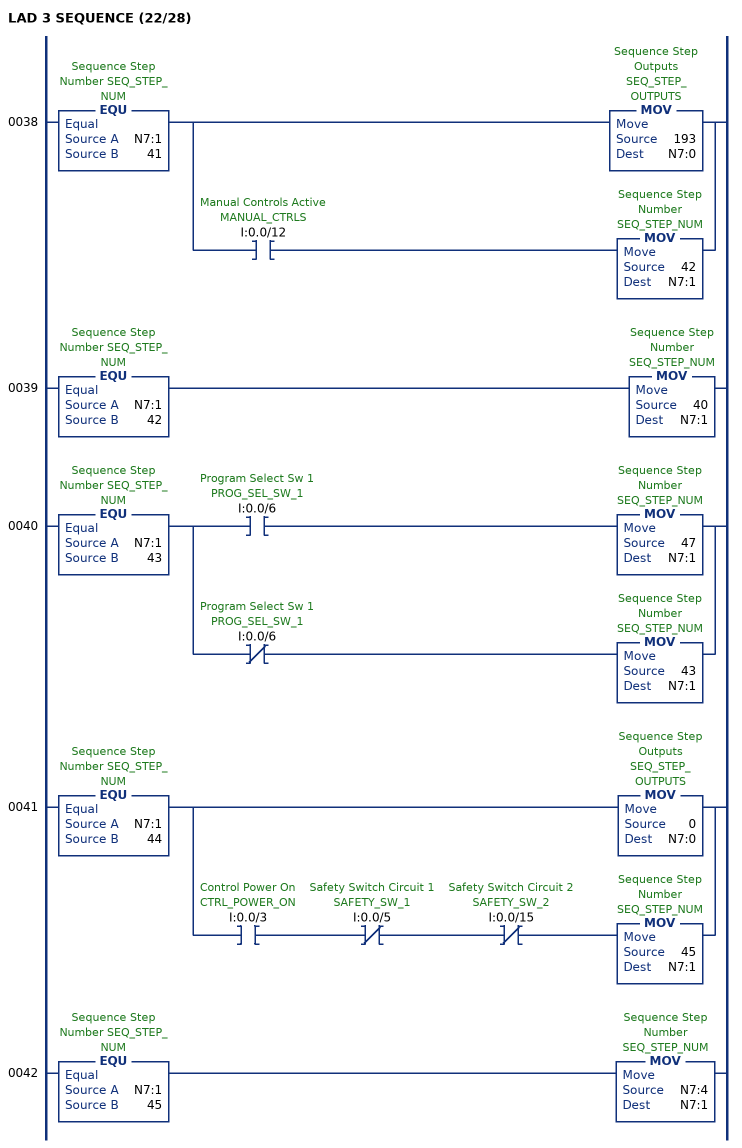
% Rung: 38 %
SOR EQU N7:1 41 BST MOV 193 N7:0 NXB XIC I:0.0/12 MOV 42 N7:1 BND EOR
%   N7:1  SEQ_STEP_NUM  "Sequence Step Number" %
%   N7:0  SEQ_STEP_OUTPUTS  "Sequence Step Outputs" %
%   I:0.0/12  MANUAL_CTRLS  "Manual Controls Active" %
% Rung: 39 %
SOR EQU N7:1 42 MOV 40 N7:1 EOR
%   N7:1  SEQ_STEP_NUM  "Sequence Step Number" %
% Rung: 40 %
SOR EQU N7:1 43 BST XIC I:0.0/6 MOV 47 N7:1 NXB XIO I:0.0/6 MOV 43 N7:1 BND EOR
%   N7:1  SEQ_STEP_NUM  "Sequence Step Number" %
%   I:0.0/6  PROG_SEL_SW_1  "Program Select Sw 1" %
% Rung: 41 %
SOR EQU N7:1 44 BST MOV 0 N7:0 NXB XIC I:0.0/3 XIO I:0.0/5 XIO I:0.0/15 MOV 45 N7:1 BND EOR
%   N7:1  SEQ_STEP_NUM  "Sequence Step Number" %
%   N7:0  SEQ_STEP_OUTPUTS  "Sequence Step Outputs" %
%   I:0.0/3  CTRL_POWER_ON  "Control Power On" %
%   I:0.0/5  SAFETY_SW_1  "Safety Switch Circuit 1" %
%   I:0.0/15  SAFETY_SW_2  "Safety Switch Circuit 2" %
% Rung: 42 %
SOR EQU N7:1 45 MOV N7:4 N7:1 EOR
%   N7:1  SEQ_STEP_NUM  "Sequence Step Number" %
%   N7:4  STORED_SEQ_STEP  "Stored Sequence Step" %

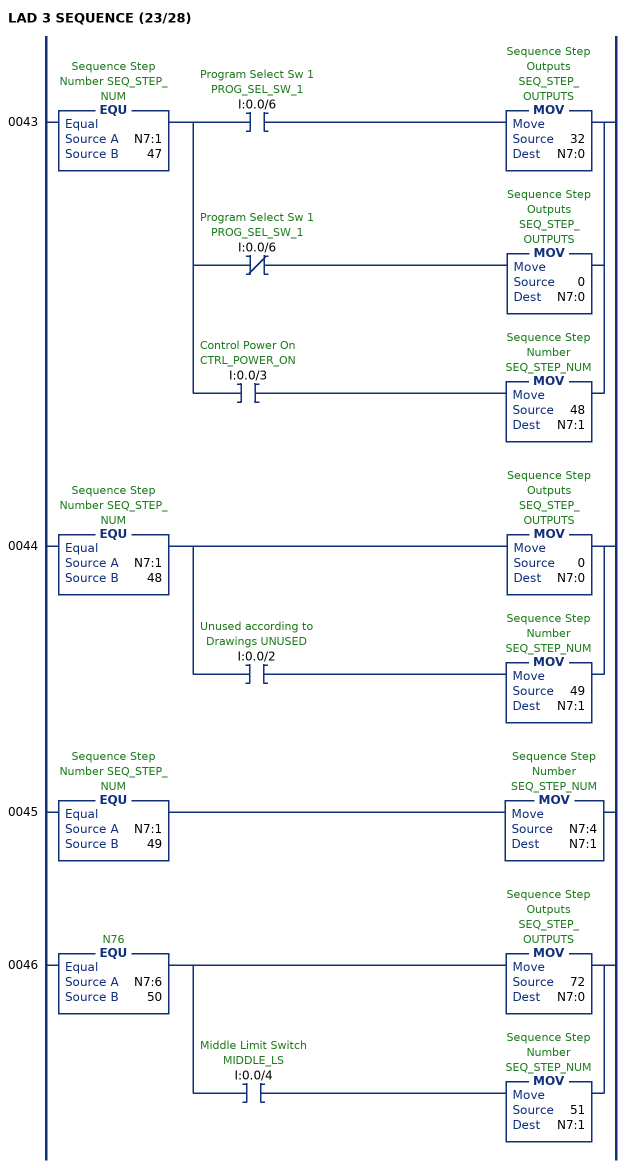
% Rung: 43 %
SOR EQU N7:1 47 BST XIC I:0.0/6 MOV 32 N7:0 NXB XIO I:0.0/6 MOV 0 N7:0 NXB XIC I:0.0/3 MOV 48 N7:1 BND EOR
%   N7:1  SEQ_STEP_NUM  "Sequence Step Number" %
%   I:0.0/6  PROG_SEL_SW_1  "Program Select Sw 1" %
%   N7:0  SEQ_STEP_OUTPUTS  "Sequence Step Outputs" %
%   I:0.0/3  CTRL_POWER_ON  "Control Power On" %
% Rung: 44 %
SOR EQU N7:1 48 BST MOV 0 N7:0 NXB XIC I:0.0/2 MOV 49 N7:1 BND EOR
%   N7:1  SEQ_STEP_NUM  "Sequence Step Number" %
%   N7:0  SEQ_STEP_OUTPUTS  "Sequence Step Outputs" %
%   I:0.0/2  UNUSED  "Unused according to Drawings" %
% Rung: 45 %
SOR EQU N7:1 49 MOV N7:4 N7:1 EOR
%   N7:1  SEQ_STEP_NUM  "Sequence Step Number" %
%   N7:4  STORED_SEQ_STEP  "Stored Sequence Step" %
% Rung: 46 %
SOR EQU N7:6 50 BST MOV 72 N7:0 NXB XIC I:0.0/4 MOV 51 N7:1 BND EOR
%   N7:6  N76 %
%   N7:0  SEQ_STEP_OUTPUTS  "Sequence Step Outputs" %
%   I:0.0/4  MIDDLE_LS  "Middle Limit Switch" %
%   N7:1  SEQ_STEP_NUM  "Sequence Step Number" %

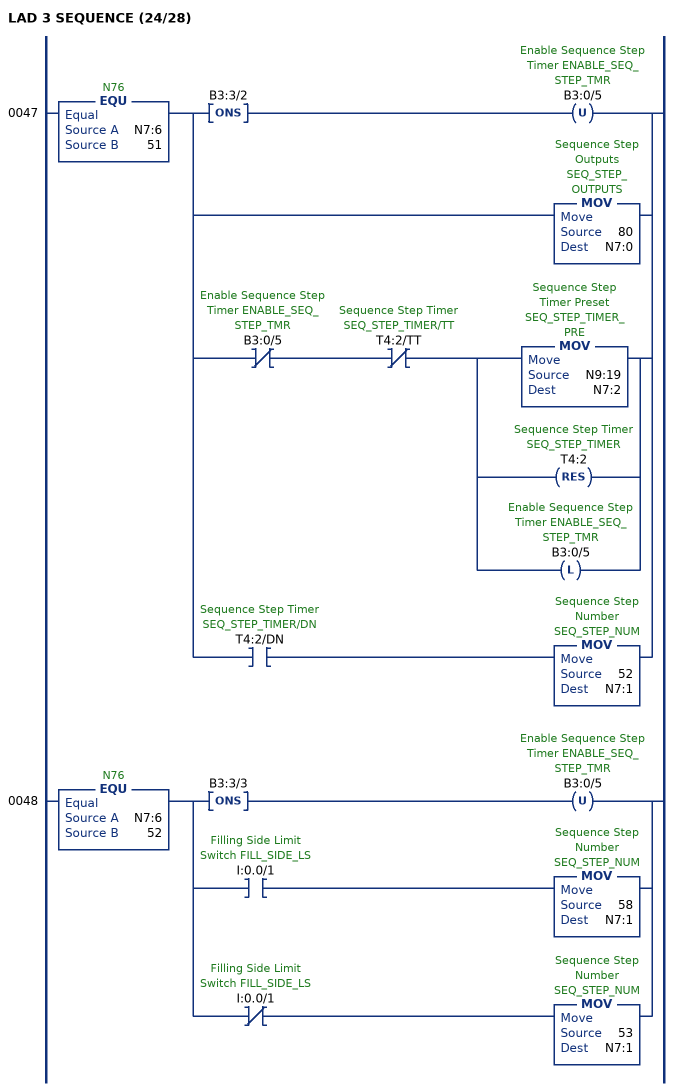
% Rung: 47 %
SOR EQU N7:6 51 BST ONS B3:3/2 OTU B3:0/5 NXB MOV 80 N7:0 NXB XIO B3:0/5 XIO T4:2/TT BST MOV N9:19 N7:2 NXB RES T4:2 NXB OTL B3:0/5 BND NXB XIC T4:2/DN MOV 52 N7:1 BND EOR
%   N7:6  N76 %
%   B3:0/5  ENABLE_SEQ_STEP_TMR  "Enable Sequence Step Timer" %
%   N7:0  SEQ_STEP_OUTPUTS  "Sequence Step Outputs" %
%   T4:2  SEQ_STEP_TIMER  "Sequence Step Timer" %
%   N7:2  SEQ_STEP_TIMER_PRE  "Sequence Step Timer Preset" %
%   N7:1  SEQ_STEP_NUM  "Sequence Step Number" %
% Rung: 48 %
SOR EQU N7:6 52 BST ONS B3:3/3 OTU B3:0/5 NXB XIC I:0.0/1 MOV 58 N7:1 NXB XIO I:0.0/1 MOV 53 N7:1 BND EOR
%   N7:6  N76 %
%   B3:0/5  ENABLE_SEQ_STEP_TMR  "Enable Sequence Step Timer" %
%   I:0.0/1  FILL_SIDE_LS  "Filling Side Limit Switch" %
%   N7:1  SEQ_STEP_NUM  "Sequence Step Number" %

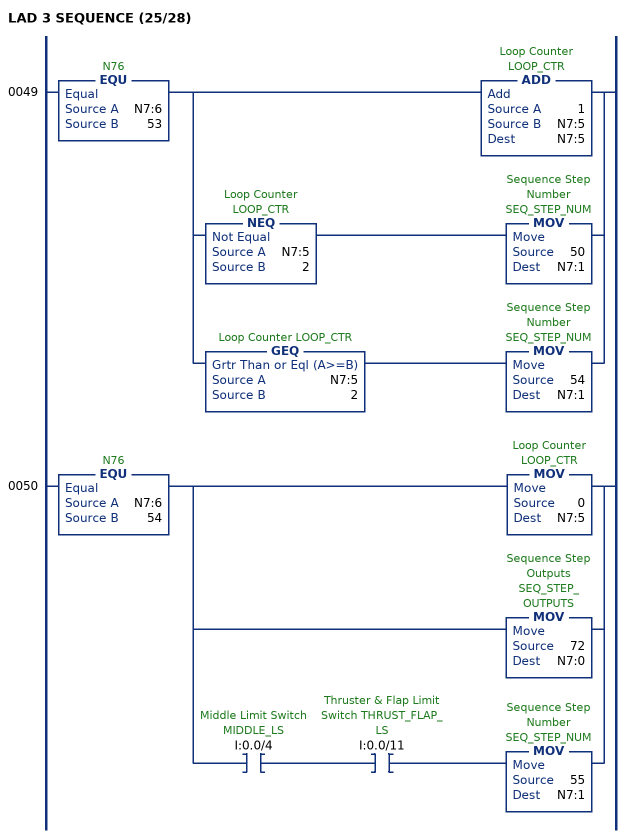
% Rung: 49 %
SOR EQU N7:6 53 BST ADD 1 N7:5 N7:5 NXB NEQ N7:5 2 MOV 50 N7:1 NXB GEQ N7:5 2 MOV 54 N7:1 BND EOR
%   N7:6  N76 %
%   N7:5  LOOP_CTR  "Loop Counter" %
%   N7:1  SEQ_STEP_NUM  "Sequence Step Number" %
% Rung: 50 %
SOR EQU N7:6 54 BST MOV 0 N7:5 NXB MOV 72 N7:0 NXB XIC I:0.0/4 XIC I:0.0/11 MOV 55 N7:1 BND EOR
%   N7:6  N76 %
%   N7:5  LOOP_CTR  "Loop Counter" %
%   N7:0  SEQ_STEP_OUTPUTS  "Sequence Step Outputs" %
%   I:0.0/4  MIDDLE_LS  "Middle Limit Switch" %
%   I:0.0/11  THRUST_FLAP_LS  "Thruster & Flap Limit Switch" %
%   N7:1  SEQ_STEP_NUM  "Sequence Step Number" %

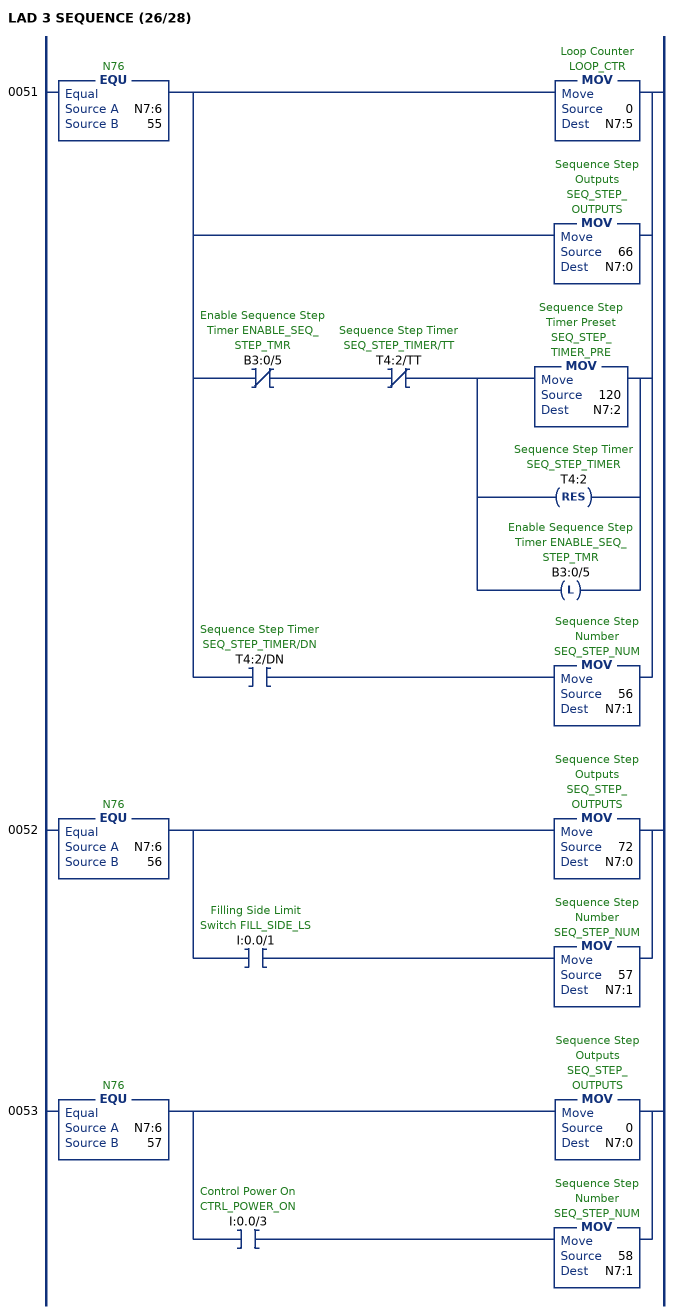
% Rung: 51 %
SOR EQU N7:6 55 BST MOV 0 N7:5 NXB MOV 66 N7:0 NXB XIO B3:0/5 XIO T4:2/TT BST MOV 120 N7:2 NXB RES T4:2 NXB OTL B3:0/5 BND NXB XIC T4:2/DN MOV 56 N7:1 BND EOR
%   N7:6  N76 %
%   N7:5  LOOP_CTR  "Loop Counter" %
%   N7:0  SEQ_STEP_OUTPUTS  "Sequence Step Outputs" %
%   B3:0/5  ENABLE_SEQ_STEP_TMR  "Enable Sequence Step Timer" %
%   T4:2  SEQ_STEP_TIMER  "Sequence Step Timer" %
%   N7:2  SEQ_STEP_TIMER_PRE  "Sequence Step Timer Preset" %
%   N7:1  SEQ_STEP_NUM  "Sequence Step Number" %
% Rung: 52 %
SOR EQU N7:6 56 BST MOV 72 N7:0 NXB XIC I:0.0/1 MOV 57 N7:1 BND EOR
%   N7:6  N76 %
%   N7:0  SEQ_STEP_OUTPUTS  "Sequence Step Outputs" %
%   I:0.0/1  FILL_SIDE_LS  "Filling Side Limit Switch" %
%   N7:1  SEQ_STEP_NUM  "Sequence Step Number" %
% Rung: 53 %
SOR EQU N7:6 57 BST MOV 0 N7:0 NXB XIC I:0.0/3 MOV 58 N7:1 BND EOR
%   N7:6  N76 %
%   N7:0  SEQ_STEP_OUTPUTS  "Sequence Step Outputs" %
%   I:0.0/3  CTRL_POWER_ON  "Control Power On" %
%   N7:1  SEQ_STEP_NUM  "Sequence Step Number" %

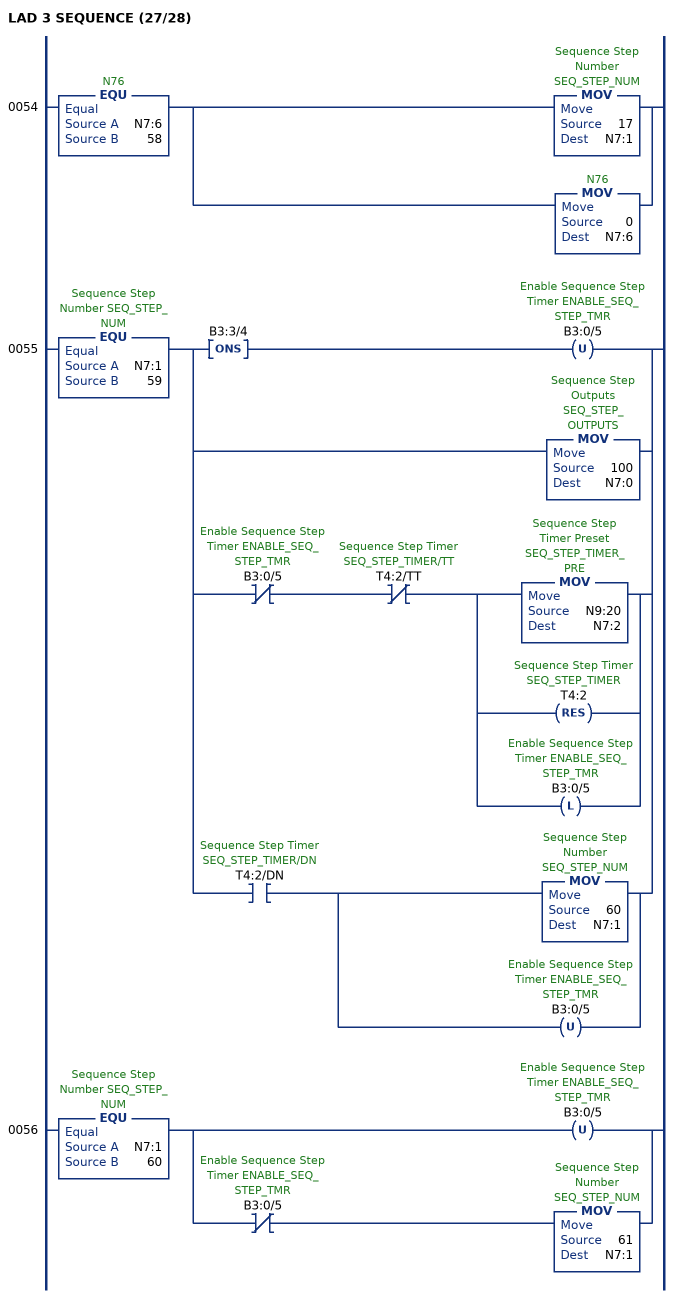
% Rung: 54 %
SOR EQU N7:6 58 BST MOV 17 N7:1 NXB MOV 0 N7:6 BND EOR
%   N7:6  N76 %
%   N7:1  SEQ_STEP_NUM  "Sequence Step Number" %
% Rung: 55 %
SOR EQU N7:1 59 BST ONS B3:3/4 OTU B3:0/5 NXB MOV 100 N7:0 NXB XIO B3:0/5 XIO T4:2/TT BST MOV N9:20 N7:2 NXB RES T4:2 NXB OTL B3:0/5 BND NXB XIC T4:2/DN BST MOV 60 N7:1 NXB OTU B3:0/5 BND BND EOR
%   N7:1  SEQ_STEP_NUM  "Sequence Step Number" %
%   B3:0/5  ENABLE_SEQ_STEP_TMR  "Enable Sequence Step Timer" %
%   N7:0  SEQ_STEP_OUTPUTS  "Sequence Step Outputs" %
%   T4:2  SEQ_STEP_TIMER  "Sequence Step Timer" %
%   N7:2  SEQ_STEP_TIMER_PRE  "Sequence Step Timer Preset" %
% Rung: 56 %
SOR EQU N7:1 60 BST OTU B3:0/5 NXB XIO B3:0/5 MOV 61 N7:1 BND EOR
%   N7:1  SEQ_STEP_NUM  "Sequence Step Number" %
%   B3:0/5  ENABLE_SEQ_STEP_TMR  "Enable Sequence Step Timer" %

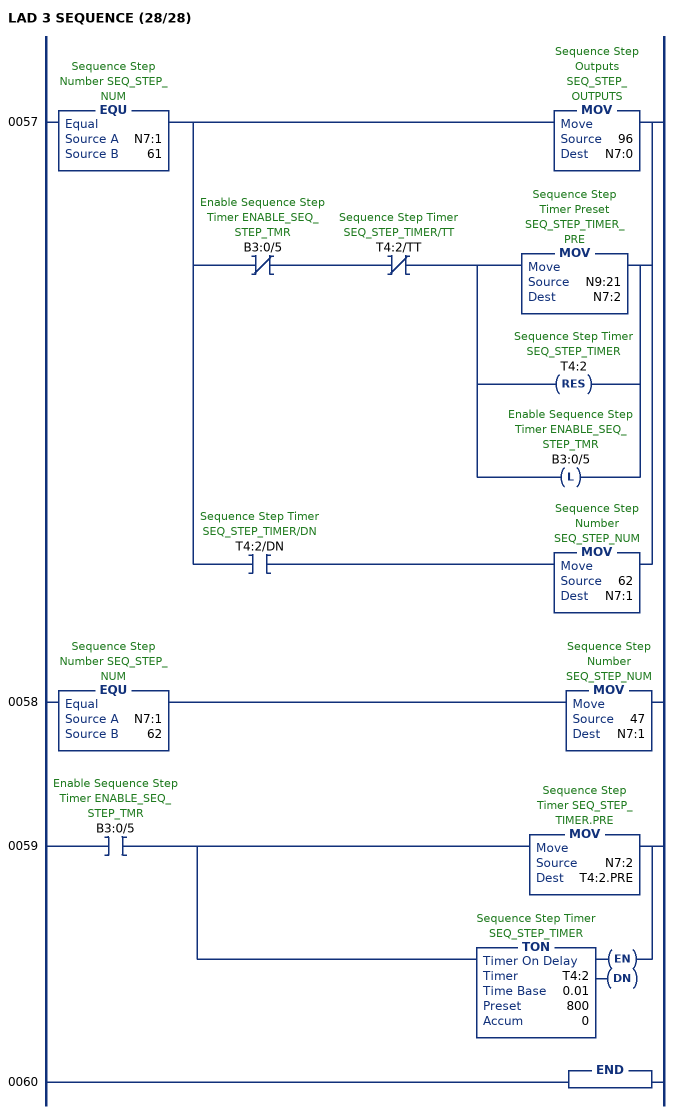
% Rung: 57 %
SOR EQU N7:1 61 BST MOV 96 N7:0 NXB XIO B3:0/5 XIO T4:2/TT BST MOV N9:21 N7:2 NXB RES T4:2 NXB OTL B3:0/5 BND NXB XIC T4:2/DN MOV 62 N7:1 BND EOR
%   N7:1  SEQ_STEP_NUM  "Sequence Step Number" %
%   N7:0  SEQ_STEP_OUTPUTS  "Sequence Step Outputs" %
%   B3:0/5  ENABLE_SEQ_STEP_TMR  "Enable Sequence Step Timer" %
%   T4:2  SEQ_STEP_TIMER  "Sequence Step Timer" %
%   N7:2  SEQ_STEP_TIMER_PRE  "Sequence Step Timer Preset" %
% Rung: 58 %
SOR EQU N7:1 62 MOV 47 N7:1 EOR
%   N7:1  SEQ_STEP_NUM  "Sequence Step Number" %
% Rung: 59 %
SOR XIC B3:0/5 BST MOV N7:2 T4:2.PRE NXB TON T4:2 0.01 800 0 BND EOR
%   B3:0/5  ENABLE_SEQ_STEP_TMR  "Enable Sequence Step Timer" %
%   N7:2  SEQ_STEP_TIMER_PRE  "Sequence Step Timer Preset" %
%   T4:2  SEQ_STEP_TIMER  "Sequence Step Timer" %
% Rung: 60 %
SOR END EOR

LADDER 4 "OUTPUTS"
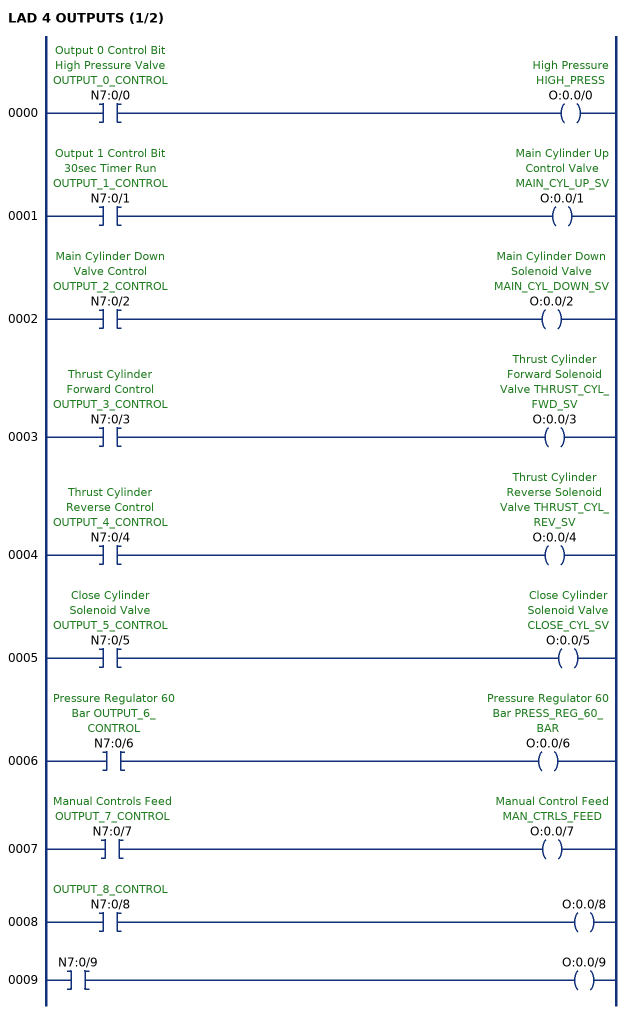
% Rung: 0 %
SOR XIC N7:0/0 OTE O:0.0/0 EOR
%   N7:0/0  OUTPUT_0_CONTROL  "Output 0 Control Bit High Pressure Valve" %
%   O:0.0/0  HIGH_PRESS  "High Pressure" %
% Rung: 1 %
SOR XIC N7:0/1 OTE O:0.0/1 EOR
%   N7:0/1  OUTPUT_1_CONTROL  "Output 1 Control Bit 30sec Timer Run" %
%   O:0.0/1  MAIN_CYL_UP_SV  "Main Cylinder Up Control Valve" %
% Rung: 2 %
SOR XIC N7:0/2 OTE O:0.0/2 EOR
%   N7:0/2  OUTPUT_2_CONTROL  "Main Cylinder Down Valve Control" %
%   O:0.0/2  MAIN_CYL_DOWN_SV  "Main Cylinder Down Solenoid Valve" %
% Rung: 3 %
SOR XIC N7:0/3 OTE O:0.0/3 EOR
%   N7:0/3  OUTPUT_3_CONTROL  "Thrust Cylinder Forward Control" %
%   O:0.0/3  THRUST_CYL_FWD_SV  "Thrust Cylinder Forward Solenoid Valve" %
% Rung: 4 %
SOR XIC N7:0/4 OTE O:0.0/4 EOR
%   N7:0/4  OUTPUT_4_CONTROL  "Thrust Cylinder Reverse Control" %
%   O:0.0/4  THRUST_CYL_REV_SV  "Thrust Cylinder Reverse Solenoid Valve" %
% Rung: 5 %
SOR XIC N7:0/5 OTE O:0.0/5 EOR
%   N7:0/5  OUTPUT_5_CONTROL  "Close Cylinder Solenoid Valve" %
%   O:0.0/5  CLOSE_CYL_SV  "Close Cylinder Solenoid Valve" %
% Rung: 6 %
SOR XIC N7:0/6 OTE O:0.0/6 EOR
%   N7:0/6  OUTPUT_6_CONTROL  "Pressure Regulator 60 Bar" %
%   O:0.0/6  PRESS_REG_60_BAR  "Pressure Regulator 60 Bar" %
% Rung: 7 %
SOR XIC N7:0/7 OTE O:0.0/7 EOR
%   N7:0/7  OUTPUT_7_CONTROL  "Manual Controls Feed" %
%   O:0.0/7  MAN_CTRLS_FEED  "Manual Control Feed" %
% Rung: 8 %
SOR XIC N7:0/8 OTE O:0.0/8 EOR
%   N7:0/8  OUTPUT_8_CONTROL %
% Rung: 9 %
SOR XIC N7:0/9 OTE O:0.0/9 EOR

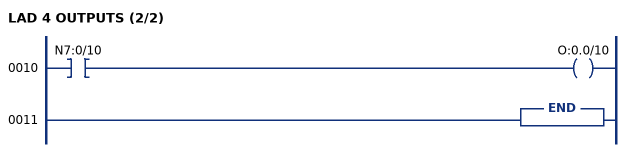
% Rung: 10 %
SOR XIC N7:0/10 OTE O:0.0/10 EOR
% Rung: 11 %
SOR END EOR

OTHER DOCUMENTED ADDRESSES
  N7:0/11  OUTPUT_11_CONTROL  "Main Motor Control"
  N7:0/12  OUTPUT_12_CONTROL  "Main Motor Delta"
  N7:0/13  OUTPUT_13_CONTROL  "Main Motor Star Control"

DATA TABLE (non-zero values as saved)
DATA T4
% .PRE .ACC %
% T4:0 % 30 0
% T4:1 % 10 0
% T4:2 % 800 0
DATA C5
% .PRE .ACC %
% C5:0 % 10000 7
DATA N7
% N7:0 % 99 22 800 0 1 0 0
DATA N9
% N9:0 % 300 100 100 100 100 30 10 800 10 40
% N9:10 % 10 20 10 10 450 40 10 10 450 200
% N9:20 % 500 200 0 0 0 0 0 0 0 0
